Yaskawa INFORM job: CLEACING-STATION-1.JBI

/JOB
//NAME CLEACING-STATION-1
//POS
///NPOS 0,0,0,0,0,2
///TOOL 0
///POSTYPE ANGLE
///ANGLE
EX00040=180.0000
EX00041=-1.0000
//INST
///DATE 2018/10/01 08:52
///ATTR SC,RW
///GROUP1 ST1
NOP
*turn
IFTHEN IN#(17)=ON
	 IMOV EX040 VJ=25.00
ENDIF
IFTHEN IN#(18)=ON
	 IMOV EX041 VJ=25.00
ENDIF
JUMP *turn IF IN#(630)=OFF
END
